Fanuc KAREL source: CNC_DYN_DISS.kl

PROGRAM T
%NOLOCKGROUP
VAR
 v0 : STRING[40]
 v1 : STRING[40]
 v2 : INTEGER
BEGIN
 CNC_DYN_DISS(v0, v1, v2)
END T
